INTERFACE I_NcAxis_HMI EXTENDS I_AxisStatus

PROPERTY Coupled : BOOL
GET
END_GET
END_PROPERTY

{attribute 'monitoring':='call'}
PROPERTY LUID : STRING  //Locally unique identifier
GET
END_GET
END_PROPERTY

PROPERTY Moving : BOOL
GET
END_GET
END_PROPERTY

{attribute 'OPC.UA.DA.Property' := '1'}
{attribute 'monitoring':='call'}
PROPERTY NcAxisName : String(31)
GET
END_GET
END_PROPERTY

END_INTERFACE

(* stored: Version 1.1.0.1, ProductVersion 3.1.4024.12
   Itf I_NcAxis_HMI: Id {97147327-7d79-065e-158d-39b7eb2c699e}
   Folder Status: Id {f4ee4c38-8e1a-0f5b-2310-696577aed203}
   Property Coupled: Id {951b5ff6-5142-4cfc-b5f6-60097a57fce4}
   Get Get: Id {02f201be-d91c-4ee4-9953-34ef4bd96129}
   Property LUID: Id {b1891b5e-8825-4dae-893a-1b6108c406e4}
   Get Get: Id {a5b9d4fd-0e70-4a5a-b4fd-bd04c01327ed}
   Property Moving: Id {be186a69-45ce-44b8-b955-199deb6bbd0b}
   Get Get: Id {90b49046-a309-41f7-b2e6-4867f58ff462}
   Property NcAxisName: Id {8db492db-8f60-4e27-bc9f-dd5bf7d4cb17}
   Get Get: Id {6c9f98d1-bd5a-4e20-9e7d-b193e18ffa50} *)
